// TIA Portal V19 export
TYPE "LEXCHANGETRAY_typeRollerVfdManualCommands"
// vfdSportsIncEnable: Bool
// vfdSportsIncReset: Bool
// sinaCommands: LBC_typeSinaSpeedManualCommands
// stored: Access Published
   STRUCT
      vfdSportsIncEnable : Bool;
      vfdSportsIncReset : Bool;
      sinaCommands : "LBC_typeSinaSpeedManualCommands";
   END_STRUCT;
END_TYPE
